FUNCTION_BLOCK InterfaceTaskExample
VAR
	_parameter : I_ParameterPosition;
	_status	   : I_ParameterPosition;
END_VAR

METHOD CyclicLogic
VAR_INPUT
END_VAR
IF _parameter = 0 OR _status = 0 THEN
	RETURN;
END_IF
_status.Position := _parameter.Position;
END_METHOD

//FB_Init is always available implicitly and it is used primarily for initialization.
//The return value is not evaluated. For a specific influence, you can also declare the
//methods explicitly and provide additional code there with the standard initialization
//code. You can evaluate the return value.
METHOD FB_Init: BOOL
VAR_INPUT
    bInitRetains: BOOL; // TRUE: the retain variables are initialized (reset warm / reset cold)
    bInCopyCode: BOOL;  // TRUE: the instance will be copied to the copy code afterward (online change)   
	Parameter : I_ParameterPosition;
	Status : I_ParameterPosition;
END_VAR
_parameter := Parameter;
_Status := Status;
END_METHOD

END_FUNCTION_BLOCK

(* stored: Version 1.1.0.1
   POU InterfaceTaskExample: Id {5dd8af2f-4322-4165-b098-9cb73464895d}, SpecialFunc None
   Method CyclicLogic: Id {36fd11a3-41e3-4c54-a02d-738df9db13a0}
   Method FB_Init: Id {a4af5ed6-f4c5-486d-88b0-3e79016590a9} *)
